FUNCTION Convert_UDINT_TO_DATE : Hresult
VAR_INPUT
	in : UDINT;
	out : REFERENCE TO DATE;
END_VAR
VAR
	converted : DATE;
END_VAR

converted := UDINT_TO_DATE(in);

IF (DATE_TO_UDINT(converted) <> in) THEN
	Convert_UDINT_TO_DATE := INCOMPATIBLE;
	RETURN;
END_IF

out := converted;

END_FUNCTION

(* stored: Version 1.1.0.1, ProductVersion 3.1.4024.12
   POU Convert_UDINT_TO_DATE: Id {bafa9e93-4c14-4b4b-bba4-1946d91334d8}, SpecialFunc None *)
